// TIA Portal V19 export
TYPE "LAF_typeDevDiagHwAddress"
TITLE = TypeDevDiagHwAdress
// This data type contains information of HW types to be evaluated. / Struktur HW-Adressen
// stored: Access Published
   STRUCT
      hwtype2 { ExternalAccessible := 'False'; ExternalVisible := 'False'; ExternalWritable := 'False'} : HW_DEVICE;   // HWTYPE = 2 (IODevice)
      hwtype5 { ExternalAccessible := 'False'; ExternalVisible := 'False'; ExternalWritable := 'False'} : HW_IO;   // HWTYPE = 5 (Submodul)
      hwtype5If { ExternalAccessible := 'False'; ExternalVisible := 'False'; ExternalWritable := 'False'} : HW_IO;   // HWTYPE = 5 (Submodul_PROFINET_Schnittstelle) / HWTYPE = 5 (Submodul_PROFINET_Interface)
   END_STRUCT;
END_TYPE
